FUNCTION_BLOCK FB_ShippingTransCV_RightSide EXTENDS FB_ActionBasic
VAR_INPUT
    xExecute    : BOOL;
    xAbort      : BOOL;
	xReset		: BOOL;
	TimeOut  	: LREAL := 60; // Unit : s
    Cylinder 	: REFERENCE TO UNI_CylinderList;
	Motor		: REFERENCE TO UNI_MotorList;
	Input		: REFERENCE TO ST_InputTable;
	OutPut		: REFERENCE TO ST_OutputTable;
	ShippingTransCVRequest_RightSide : BOOL;
	RobotStatus	: ST_StatusBasic;		// robot Service 
END_VAR
VAR_OUTPUT
	xAborted : BOOL;
    iErrorID : INT;
    ErrorMsg : STRING;
END_VAR
VAR
	// model setting 
	StateBehaviour   : CBML.ETrigATo;
    CurrentPosition : ST_PositionTable;
	fbExecuteEdgeDetect :FB_EdgeDetect;
	Reset_Rtrig 	:R_TRIG;
	uiCyclicStep    : UINT := 0;
	
	//Timer
	TON_DelayArrivedDetect	: TON;
	TON_TransCVAllowDelay	: TON;
END_VAR

THIS^.IBehaviourModel := StateBehaviour;

StateBehaviour(xExecute := xExecute,
              xAbort := xAbort OR fbExecuteEdgeDetect.xFallingEdge,
              udiTimeOut := LREAL_TO_UDINT( TimeOut*1000000),
              xDone => xDone,
              xBusy => xBusy,
              xError => xError,
              xAborted => xAborted);
			  
//Make sure that C# turns off execute to shut down the service
fbExecuteEdgeDetect(xInput :=xExecute);
  
//Error Msg
iErrorID := StateBehaviour._model.iErrorID;
ErrorMsg := M_GetErrorMsg(xErrorID := iErrorID);

//Reset
Reset_Rtrig(CLK:= xReset);
IF Reset_Rtrig.Q THEN
	StateBehaviour.ResetModel(xCommit:=xReset);
END_IF

//Action
A00_BaseUnit();

ACTION A00_BaseUnit:
TON_DelayArrivedDetect(PT:=T#1S);
TON_TransCVAllowDelay(PT :=T#1S);
END_ACTION

METHOD CleanupAction
VAR_INPUT
    xAbortProposed : BOOL;
    iErrorIDProposed: INT;
END_VAR
VAR_OUTPUT
    xComplete : BOOL := TRUE;
    xAbort: BOOL := xAbortProposed;
 	iErrorID : INT := iErrorIDProposed;
END_VAR
END_METHOD

METHOD CyclicAction
VAR_INPUT
    itfTimingController : CBML.ITimingController;
END_VAR
VAR_OUTPUT
    xComplete : BOOL := TRUE;
    iErrorID : INT := 0;
END_VAR
xComplete := FALSE;


CASE uiCyclicStep OF 
	0:	// robot status , send allow signal
		IF ShippingTransCVRequest_RightSide AND NOT RobotStatus.Busy THEN
			TON_TransCVAllowDelay.IN := TRUE;
			OutPut.bShippingTransCV_Rightside_Allow := TRUE;
		END_IF
		IF TON_TransCVAllowDelay.Q THEN
			OutPut.bShippingTransCV_Rightside_Allow := FALSE;
			uiCyclicStep := 100;
		END_IF

	100:	//check HansLaser cancel signal
		TON_TransCVAllowDelay.IN := FALSE;
		IF NOT Input.bShippingTransCV_Rightside_Arrived THEN 
			xComplete := TRUE;
		END_IF
END_CASE

IF Input.bHansLaserMachineError THEN
	iErrorID := 10;
END_IF
END_METHOD

METHOD ExitAction
VAR_INPUT
    xAfterCleanup : BOOL;
    xInCopyCode : BOOL;
END_VAR
END_METHOD

METHOD M_GetErrorMsg : T_MaxString
VAR_INPUT
	xErrorID: INT;
END_VAR

VAR
	
END_VAR
CASE xErrorID OF
	0:
		M_GetErrorMsg := 'No Error';
	1:
		M_GetErrorMsg := 'FB_ShippingTransCV_RightSide ErrorID 1: Action time out';
///
	10:
		M_GetErrorMsg := 'FB_ShippingTransCV_RightSide ErrorID 10: HansLaser Machine Error';
	11:
		M_GetErrorMsg := 'FB_ShippingTransCV_RightSide ErrorID 11: Wrong Command , TransCV not IntargetPosition';
END_CASE
END_METHOD

METHOD ResetAction
VAR_OUTPUT
    xComplete : BOOL := TRUE;
END_VAR
xComplete := FALSE;

ShippingTransCVRequest_RightSide 		:= FALSE;
OutPut.bShippingTransCV_Rightside_Allow := FALSE;

TON_DelayArrivedDetect.IN := FALSE;
TON_TransCVAllowDelay.IN := FALSE;

uiCyclicStep := 0;

xComplete := TRUE;
END_METHOD

METHOD StartAction
VAR_OUTPUT
    xComplete : BOOL := TRUE;
	iErrorID : INT := 0;
END_VAR
xComplete := FALSE;

ShippingTransCVRequest_RightSide 		:= FALSE;
OutPut.bShippingTransCV_Rightside_Allow := FALSE;

uiCyclicStep := 0;

TON_DelayArrivedDetect.IN := FALSE;
TON_TransCVAllowDelay.IN := FALSE;




IF Input.bHansLaserMachineError THEN
	iErrorID := 10;
END_IF

IF NOT Input.bShippingTransCV_Rightside_Arrived THEN
	iErrorID := 11;
END_IF

xComplete := TRUE;
END_METHOD

END_FUNCTION_BLOCK

(* stored: Version 1.1.0.1, ProductVersion 3.1.4024.13
   POU FB_ShippingTransCV_RightSide: Id {8a62b2be-7f93-4080-8aa4-d8dd8a7f8439}, SpecialFunc None
   Folder Action: Id {49f5d86b-14f7-4daf-b5e7-2843476bd95e}
   Action A00_BaseUnit: Id {b93c2a8d-98ba-4b03-b46f-780d5f35ffe8}
   Method CleanupAction: Id {f3466de0-49cf-4aed-8f55-776a8c394f28}
   Method CyclicAction: Id {3291e4b4-4f35-4936-9d05-2b504294a2d0}
   Method ExitAction: Id {47ae62b6-b2a8-4da4-979f-a3f32c007581}
   Method M_GetErrorMsg: Id {a417501a-8ada-49e8-bd18-9bd59443c0d6}
   Method ResetAction: Id {3265f16f-fb2e-46a7-991c-1b0cd9057161}
   Method StartAction: Id {52b5f349-c710-40a8-b540-0b06a0d9a452} *)
